Fanuc KAREL source: ko00037.KL

-- PROVISIONAL review KL for V1013-1; original PC SHA256 d5b8966fba0e6a77ce22ddcc839bffdacede860835f4f9981e48d524cb05f54d
-- Incomplete behavior may be omitted. Consult companion uncertainty JSON. Do not deploy.
PROGRAM KO00037
%NOLOCKGROUP
BEGIN
  -- UNRESOLVED_PC offsets 5-12; opcodes 9D,23
  -- UNRESOLVED_PC offsets 17-69; opcodes 27,27,49,7E,AD,27,49,7E,AD,22,31,7E,4A
  -- UNRESOLVED_PC offsets 74-78; opcodes 7F
END KO00037
